// TIA Portal V20 export
VAR_GLOBAL   // PLC tag table "Constantes del Tracking"
END_VAR
VAR_GLOBAL CONSTANT   // user constants
   CTE_Long_Accesos : UInt := 42;   // Longitud de la Estructura de Accesos a Recintos
   CTE_Long_VIMaquina : UInt := 16;   // Longitud del Estado VI Maquina
   CTE_Long_VIMesa : UInt := 16;   // Longitud del Estado VI Mesa
   CTE_LongFIFO : UInt := 4;
   CTE_NDB_EstadoVIMaquina : UInt := 904;   // Num DB del Estado VI Maquina
   CTE_NDB_EstadoVIMesa : UInt := 900;   // Num DB del Estado VI Mesa
   CTE_NDB_Accesos : UInt := 918;   // Num DB de los Datos de Accesos a Recintos
   CTE_NumMesas_Accesos : UInt := 19;   // Maximo Numero de Mesas de Accesos a Recintos
   CTE_NDB_ErroresArmarios : UInt := 860;
END_VAR
